FUNCTION_BLOCK FB_SendIampTemp_Left
VAR_INPUT
	Iamp_Temp : LREAL;
END_VAR
VAR_OUTPUT
END_VAR
VAR
	TxMessage : EXTCANQUEUE;
	i : INT;
	Iamp_Temp_Values : ARRAY[0..1] OF BYTE;
END_VAR
VAR_IN_OUT
	CAN_OUTPUTS_Left : CANTXQUEUESTRUCT_E_32;
	CAN_INPUTS_Left : CANRXQUEUESTRUCT_E_32;
END_VAR

Iamp_Temp_Values[1] := INT_TO_BYTE(LREAL_TO_INT(Iamp_Temp) AND 16#FF);
Iamp_Temp_Values[0] := INT_TO_BYTE(SHR(LREAL_TO_INT(Iamp_Temp), 8) AND 16#FF);


TxMessage.cobId := 1600;
TxMessage.length := 2;
FOR i := 0 TO 1 DO 
		TxMessage.data[i] := Iamp_Temp_Values[i];
END_FOR
CAN_OUTPUTS_Left.TxMessages[14] := TxMessage;
//CAN_OUTPUTS.NoOfTxMessages := 1;

END_FUNCTION_BLOCK

(* stored: Version 1.1.0.1
   POU FB_SendIampTemp_Left: Id {06569dc7-df18-4bd0-bcb7-189062d8240b}, SpecialFunc None *)
